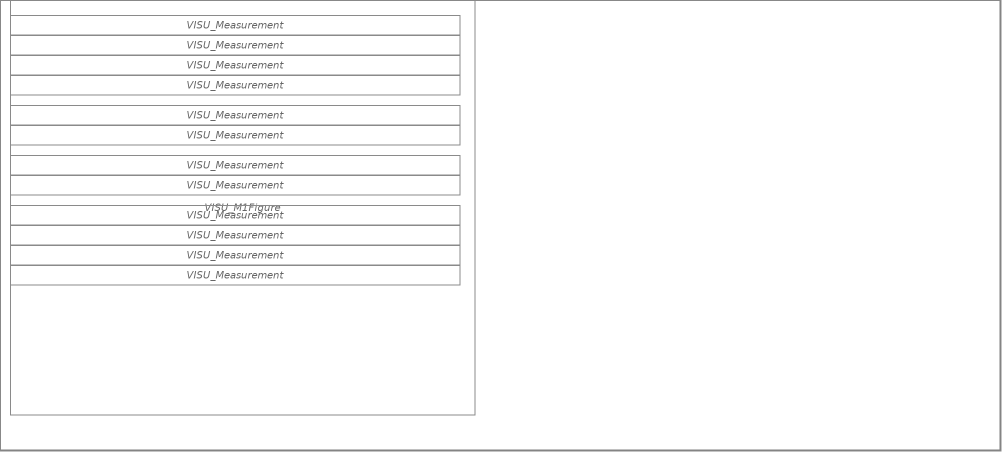
VISUALIZATION VISU_M1FullFigure  // 1002x452
VAR_IN_OUT
	ref : M1;
    widget : M1Widget;
END_VAR
    Rectangle (0,0 1000x450)
    Frame (10,0 465x415)
        shows VISU_M1Figure(ref := ref, widget := widget)
    Frame (10,15 450x20)
        shows VISU_Measurement(widget := widget.pneumaticSupplyPressure)
    Frame (10,35 450x20)
        shows VISU_Measurement(widget := widget.inclinometer.voltageMeasurement)
    Frame (10,55 450x20)
        shows VISU_Measurement(widget := widget.inclinometer.elevation)
    Frame (10,105 450x20)
        shows VISU_Measurement(widget := widget.radialSupport.regulatorPressure)
    Frame (10,125 450x20)
        shows VISU_Measurement(widget := widget.radialSupport.mirrorPressure)
    Frame (10,175 450x20)
        shows VISU_Measurement(widget := widget.axialSupport.mirrorPressure)
    Frame (10,155 450x20)
        shows VISU_Measurement(widget := widget.axialSupport.regulatorPressure)
    Frame (10,225 450x20)
        shows VISU_Measurement(widget := widget.axialSupport.mirrorNorthEastForce)
    Frame (10,205 450x20)
        shows VISU_Measurement(widget := widget.axialSupport.mirrorSouthForce)
    Frame (10,245 450x20)
        shows VISU_Measurement(widget := widget.axialSupport.mirrorNorthWestForce)
    Frame (10,265 450x20)
        shows VISU_Measurement(widget := widget.axialSupport.mirrorAverageForce)
    Frame (10,75 450x20)
        shows VISU_Measurement(widget := widget.accelerometerAngle)
END_VISUALIZATION

(* stored: Version 1.1.0.1, ProductVersion 3.1.4019.2
   Visu VISU_M1FullFigure: Id {7189ae92-e102-48c6-b658-b28291965e93} *)
